// TIA Portal V18 export
// export: Created 2026-06-20T23:26:23.319602Z, ExportSetting WithDefaults
TextList "TL_Canh_Bao_Mixing"  ListRange=Decimal, Comment="Cảnh báo Mixing"
  TextListEntry   EntryType=SingleValue, Text="[AN TOÀN] Không có cảnh báo"
  TextListEntry   EntryType=SingleValue, From=1, To=1, Text="[DOSING] Van mở nhưng lưu lượng không tăng"
  TextListEntry   EntryType=SingleValue, From=2, To=2, Text="[SETPOINT] Giá trị setpoint không hợp lệ"
  TextListEntry   EntryType=SingleValue, From=3, To=3, Text="[KHÓA AN TOÀN] Dry run hoặc liên động bảo vệ"
  TextListEntry   EntryType=SingleValue, From=4, To=4, Text="[ESTOP ACTIVE] Dừng khẩn đang được chốt"
